FUNCTION_BLOCK basicInfluentFeedLogic (* Basic Function Block Type *)
  (* Standard: 61499-2 *)
  (* Version 0.0, 13/09/2026, Template *)
  PACKAGE Hidryco.HidrycoLib;
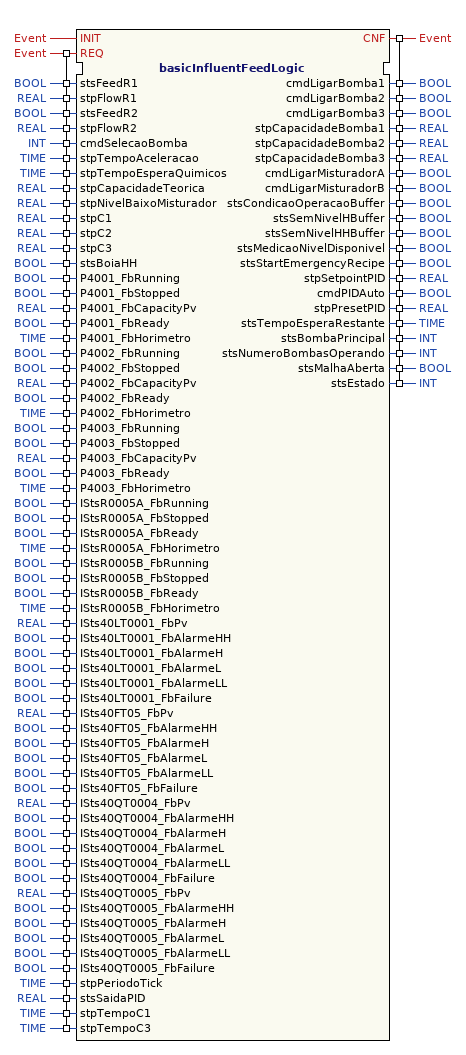
  EVENT_INPUT
    INIT;
    REQ WITH stsFeedR1, stpFlowR1, stsFeedR2, stpFlowR2, cmdSelecaoBomba, stpTempoAceleracao, stpTempoEsperaQuimicos, stpCapacidadeTeorica, stpNivelBaixoMisturador, stpC1, stpC2, stpC3, stsBoiaHH, P4001_FbRunning, P4001_FbStopped, P4001_FbCapacityPv, P4001_FbReady, P4001_FbHorimetro, P4002_FbRunning, P4002_FbStopped, P4002_FbCapacityPv, P4002_FbReady, P4002_FbHorimetro, P4003_FbRunning, P4003_FbStopped, P4003_FbCapacityPv, P4003_FbReady, P4003_FbHorimetro, IStsR0005A_FbRunning, IStsR0005A_FbStopped, IStsR0005A_FbReady, IStsR0005A_FbHorimetro, IStsR0005B_FbRunning, IStsR0005B_FbStopped, IStsR0005B_FbReady, IStsR0005B_FbHorimetro, ISts40LT0001_FbPv, ISts40LT0001_FbAlarmeHH, ISts40LT0001_FbAlarmeH, ISts40LT0001_FbAlarmeL, ISts40LT0001_FbAlarmeLL, ISts40LT0001_FbFailure, ISts40FT05_FbPv, ISts40FT05_FbAlarmeHH, ISts40FT05_FbAlarmeH, ISts40FT05_FbAlarmeL, ISts40FT05_FbAlarmeLL, ISts40FT05_FbFailure, ISts40QT0004_FbPv, ISts40QT0004_FbAlarmeHH, ISts40QT0004_FbAlarmeH, ISts40QT0004_FbAlarmeL, ISts40QT0004_FbAlarmeLL, ISts40QT0004_FbFailure, ISts40QT0005_FbPv, ISts40QT0005_FbAlarmeHH, ISts40QT0005_FbAlarmeH, ISts40QT0005_FbAlarmeL, ISts40QT0005_FbAlarmeLL, ISts40QT0005_FbFailure, stpPeriodoTick, stsSaidaPID, stpTempoC1, stpTempoC3; (* Normal Execution Request *)
  END_EVENT
  EVENT_OUTPUT
    CNF WITH cmdLigarBomba1, cmdLigarBomba2, cmdLigarBomba3, stpCapacidadeBomba1, stpCapacidadeBomba2, stpCapacidadeBomba3, cmdLigarMisturadorA, cmdLigarMisturadorB, stsCondicaoOperacaoBuffer, stsSemNivelHBuffer, stsSemNivelHHBuffer, stsMedicaoNivelDisponivel, stsStartEmergencyRecipe, stpSetpointPID, cmdPIDAuto, stpPresetPID, stsTempoEsperaRestante, stsBombaPrincipal, stsNumeroBombasOperando, stsMalhaAberta, stsEstado; (* Execution Confirmation *)
  END_EVENT
  VAR_INPUT
    stsFeedR1 : BOOL;
    stpFlowR1 : REAL;
    stsFeedR2 : BOOL;
    stpFlowR2 : REAL;
    cmdSelecaoBomba : INT;
    stpTempoAceleracao : TIME; (* Espera antes de controlar as duas bombas juntas *)
    stpTempoEsperaQuimicos : TIME; (* Espera para reiniciar após pH e condutividade normalizarem *)
    stpCapacidadeTeorica : REAL; (* Vazão nominal, para a malha aberta *)
    stpNivelBaixoMisturador : REAL; (* Bloqueio para misturadores *)
    stpC1 : REAL;
    stpC2 : REAL;
    stpC3 : REAL;
    stsBoiaHH : BOOL;
    P4001_FbRunning : BOOL;
    P4001_FbStopped : BOOL;
    P4001_FbCapacityPv : REAL;
    P4001_FbReady : BOOL;
    P4001_FbHorimetro : TIME;
    P4002_FbRunning : BOOL;
    P4002_FbStopped : BOOL;
    P4002_FbCapacityPv : REAL;
    P4002_FbReady : BOOL;
    P4002_FbHorimetro : TIME;
    P4003_FbRunning : BOOL;
    P4003_FbStopped : BOOL;
    P4003_FbCapacityPv : REAL;
    P4003_FbReady : BOOL;
    P4003_FbHorimetro : TIME;
    IStsR0005A_FbRunning : BOOL;
    IStsR0005A_FbStopped : BOOL;
    IStsR0005A_FbReady : BOOL;
    IStsR0005A_FbHorimetro : TIME;
    IStsR0005B_FbRunning : BOOL;
    IStsR0005B_FbStopped : BOOL;
    IStsR0005B_FbReady : BOOL;
    IStsR0005B_FbHorimetro : TIME;
    ISts40LT0001_FbPv : REAL;
    ISts40LT0001_FbAlarmeHH : BOOL;
    ISts40LT0001_FbAlarmeH : BOOL;
    ISts40LT0001_FbAlarmeL : BOOL;
    ISts40LT0001_FbAlarmeLL : BOOL;
    ISts40LT0001_FbFailure : BOOL;
    ISts40FT05_FbPv : REAL;
    ISts40FT05_FbAlarmeHH : BOOL;
    ISts40FT05_FbAlarmeH : BOOL;
    ISts40FT05_FbAlarmeL : BOOL;
    ISts40FT05_FbAlarmeLL : BOOL;
    ISts40FT05_FbFailure : BOOL;
    ISts40QT0004_FbPv : REAL;
    ISts40QT0004_FbAlarmeHH : BOOL;
    ISts40QT0004_FbAlarmeH : BOOL;
    ISts40QT0004_FbAlarmeL : BOOL;
    ISts40QT0004_FbAlarmeLL : BOOL;
    ISts40QT0004_FbFailure : BOOL;
    ISts40QT0005_FbPv : REAL;
    ISts40QT0005_FbAlarmeHH : BOOL;
    ISts40QT0005_FbAlarmeH : BOOL;
    ISts40QT0005_FbAlarmeL : BOOL;
    ISts40QT0005_FbAlarmeLL : BOOL;
    ISts40QT0005_FbFailure : BOOL;
    stpPeriodoTick : TIME;
    stsSaidaPID : REAL;
    stpTempoC1 : TIME;
    stpTempoC3 : TIME;
  END_VAR
  VAR_OUTPUT
    cmdLigarBomba1 : BOOL;
    cmdLigarBomba2 : BOOL;
    cmdLigarBomba3 : BOOL;
    stpCapacidadeBomba1 : REAL;
    stpCapacidadeBomba2 : REAL;
    stpCapacidadeBomba3 : REAL;
    cmdLigarMisturadorA : BOOL;
    cmdLigarMisturadorB : BOOL;
    stsCondicaoOperacaoBuffer : BOOL; (* Operating condition da fase Feed, nos dois reatores. FALSE quando o buffer não pode alimentar *)
    stsSemNivelHBuffer : BOOL;
    stsSemNivelHHBuffer : BOOL;
    stsMedicaoNivelDisponivel : BOOL;
    stsStartEmergencyRecipe : BOOL;
    stpSetpointPID : REAL;
    cmdPIDAuto : BOOL;
    stpPresetPID : REAL;
    stsTempoEsperaRestante : TIME;
    stsBombaPrincipal : INT;
    stsNumeroBombasOperando : INT;
    stsMalhaAberta : BOOL;
    stsEstado : INT;
  END_VAR
  VAR
    iEstado : INT;
    idxDuty1 : INT;
    idxDuty2 : INT;
    tEsperaQuim : TIME;
    tAcel : TIME;
    tC1 : TIME;
    tC3 : TIME;
    bQuimOkAnt : BOOL;
    rSaida : REAL;
  END_VAR
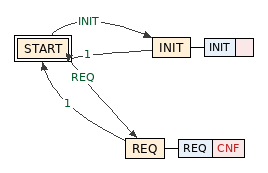
  EC_STATES
    START; (* Initial State *)
    INIT : INIT;
    REQ : REQ -> CNF;
  END_STATES
  EC_TRANSITIONS
    START TO INIT := INIT;
    INIT TO START := 1;
    START TO REQ := REQ;
    REQ TO START := 1;
  END_TRANSITIONS
  ALGORITHM INIT IN ST: (* Initialization algorithm *)
iEstado := 0;
idxDuty1 := 0;
idxDuty2 := 0;
tEsperaQuim := stpTempoEsperaQuimicos;
tAcel := stpTempoAceleracao;
tC1 := stpTempoC1;
tC3 := stpTempoC3;
bQuimOkAnt := FALSE;
rSaida := 0.0;
cmdLigarBomba1 := FALSE; cmdLigarBomba2 := FALSE; cmdLigarBomba3 := FALSE;
stpCapacidadeBomba1 := 0.0; stpCapacidadeBomba2 := 0.0; stpCapacidadeBomba3 := 0.0;
cmdLigarMisturadorA := FALSE; cmdLigarMisturadorB := FALSE;
stsCondicaoOperacaoBuffer := FALSE;
stsSemNivelHBuffer := TRUE;
stsSemNivelHHBuffer := TRUE;
stsMedicaoNivelDisponivel := FALSE;
stsStartEmergencyRecipe := FALSE;
stpSetpointPID := 0.0;
cmdPIDAuto := FALSE;
stpPresetPID := 0.0;
stsTempoEsperaRestante := T#0s;
stsBombaPrincipal := 0;
stsNumeroBombasOperando := 0;
stsMalhaAberta := FALSE;
stsEstado := 0;

;
  END_ALGORITHM
  ALGORITHM REQ IN ST: (* Normally executed algorithm *)
  VAR_TEMP
    bFeedAtivo : BOOL;
    bQuimOk : BOOL;
    bBombaDisp : BOOL;
    bVazaoLL : BOOL;
    bReadyD1 : BOOL;
    bReadyD2 : BOOL;
    rSpBruto : REAL;
    nLigadas : INT;
    idxCand : INT;
    tMenor : TIME;
  END_VAR
stsSemNivelHBuffer := NOT ISts40LT0001_FbAlarmeH;
stsSemNivelHHBuffer := NOT stsBoiaHH;
stsMedicaoNivelDisponivel := NOT ISts40LT0001_FbFailure;
stsStartEmergencyRecipe := ISts40LT0001_FbAlarmeHH
AND NOT ISts40LT0001_FbFailure;
(*------------------------------------------------------------------
2. QUÍMICOS — narrativa 2.2, 2.3.6 e 2.3.7
pH ou condutividade fora de faixa, ou falha de medição de
qualquer um dos dois, param a alimentação.
Temporizador de retomada: conta apenas com AMBOS dentro da
faixa. Qualquer saída de faixa rearma do zero.
------------------------------------------------------------------*)
bQuimOk := NOT ISts40QT0005_FbAlarmeL AND NOT ISts40QT0005_FbAlarmeH
AND NOT ISts40QT0004_FbAlarmeL AND NOT ISts40QT0004_FbAlarmeH
AND NOT ISts40QT0005_FbFailure AND NOT ISts40QT0004_FbFailure;
IF bQuimOk THEN
	IF NOT bQuimOkAnt THEN
		tEsperaQuim := stpTempoEsperaQuimicos; (* borda: arma *)
	ELSIF tEsperaQuim > stpPeriodoTick THEN
		tEsperaQuim := tEsperaQuim - stpPeriodoTick;
	ELSE
		tEsperaQuim := T#0s; (* expirou *)
	END_IF;
ELSE
	tEsperaQuim := stpTempoEsperaQuimicos; (* rearma *)
END_IF;
bQuimOkAnt := bQuimOk;
stsTempoEsperaRestante := tEsperaQuim;
(*------------------------------------------------------------------
3. BOMBAS RODANDO E LL DE VAZÃO
O atraso do alarme é feito pelo bloco de sensor. Aqui só a
supressão: com bomba parada a vazão é zero por definição, e o
alarme não pode bloquear a alimentação.
------------------------------------------------------------------*)
nLigadas := 0;
IF P4001_FbRunning THEN nLigadas := nLigadas + 1; END_IF;
IF P4002_FbRunning THEN nLigadas := nLigadas + 1; END_IF;
IF P4003_FbRunning THEN nLigadas := nLigadas + 1; END_IF;
stsNumeroBombasOperando := nLigadas;
bVazaoLL := (nLigadas > 0)
AND ISts40FT05_FbAlarmeLL
AND NOT ISts40FT05_FbFailure;
(*------------------------------------------------------------------
4. DISPONIBILIDADE — narrativa 1.4.2
------------------------------------------------------------------*)
bBombaDisp := P4001_FbReady OR P4002_FbReady OR P4003_FbReady;
(*------------------------------------------------------------------
5. CONDIÇÃO DE OPERAÇÃO DO BUFFER
Vai para a operating condition da fase Feed dos dois reatores.
Narrativa 2.2: a alimentação para em LL de nível, pH fora de
faixa e condutividade fora de faixa.
------------------------------------------------------------------*)
stsCondicaoOperacaoBuffer := bBombaDisp
AND bQuimOk
AND (tEsperaQuim = T#0s)
AND NOT ISts40LT0001_FbAlarmeLL
AND NOT ISts40LT0001_FbFailure
AND NOT bVazaoLL;
(*------------------------------------------------------------------
6. SETPOINT DE VAZÃO — narrativa 2.2 e 3.2.1
O Nereda envia m³/h; o PI converte em capacidade.
Apenas uma fase Feed pode estar em RUN por vez.
------------------------------------------------------------------*)
bFeedAtivo := stsFeedR1 OR stsFeedR2;
IF stsFeedR1 THEN rSpBruto := stpFlowR1;
ELSIF stsFeedR2 THEN rSpBruto := stpFlowR2;
ELSE rSpBruto := 0.0;
END_IF;
IF rSpBruto < 0.0 THEN rSpBruto := 0.0; END_IF;
stpSetpointPID := rSpBruto;
(*------------------------------------------------------------------
7. ESCOLHA DAS BOMBAS — narrativa 1.4.9
idxCand = próxima candidata: disponível, ainda não comandada,
de MENOR horímetro (FbHorimetro = tempo de operação).
Em modo fixo, a candidata é a bomba escolhida pelo operador.
------------------------------------------------------------------*)
idxCand := 0;
tMenor := T#999999s;
IF cmdSelecaoBomba = 1 THEN
IF P4001_FbReady AND (idxDuty1 <> 1) AND (idxDuty2 <> 1) THEN idxCand := 1; END_IF;
ELSIF cmdSelecaoBomba = 2 THEN
IF P4002_FbReady AND (idxDuty1 <> 2) AND (idxDuty2 <> 2) THEN idxCand := 2; END_IF;
ELSIF cmdSelecaoBomba = 3 THEN
IF P4003_FbReady AND (idxDuty1 <> 3) AND (idxDuty2 <> 3) THEN idxCand := 3; END_IF;
ELSE
IF P4001_FbReady AND (idxDuty1 <> 1) AND (idxDuty2 <> 1)
AND (P4001_FbHorimetro <= tMenor) THEN
idxCand := 1; tMenor := P4001_FbHorimetro;
END_IF;
IF P4002_FbReady AND (idxDuty1 <> 2) AND (idxDuty2 <> 2)
AND (P4002_FbHorimetro < tMenor) THEN
idxCand := 2; tMenor := P4002_FbHorimetro;
END_IF;
IF P4003_FbReady AND (idxDuty1 <> 3) AND (idxDuty2 <> 3)
AND (P4003_FbHorimetro < tMenor) THEN
idxCand := 3; tMenor := P4003_FbHorimetro;
END_IF;
END_IF;
(* Disponibilidade das bombas atualmente comandadas *)
bReadyD1 := FALSE;
CASE idxDuty1 OF
1: bReadyD1 := P4001_FbReady;
2: bReadyD1 := P4002_FbReady;
3: bReadyD1 := P4003_FbReady;
END_CASE;
bReadyD2 := FALSE;
CASE idxDuty2 OF
1: bReadyD2 := P4001_FbReady;
2: bReadyD2 := P4002_FbReady;
3: bReadyD2 := P4003_FbReady;
END_CASE;
stsBombaPrincipal := idxDuty1;
(*------------------------------------------------------------------
8. MÁQUINA DE ESTADOS — narrativa 2.2
0 Parado · 1 Partindo · 2 Uma bomba · 3 Sobe (C2)
4 Duas bombas · 5 Desce · 6 Parando
Na partida não há capacidade fixa: o PI assume desde o início e
a rampa do inversor cuida do transitório. C2 é usado apenas na
transição de uma para duas bombas.
------------------------------------------------------------------*)
CASE iEstado OF
0: (*--- PARADO ---*)
idxDuty1 := 0; idxDuty2 := 0;
cmdPIDAuto := FALSE; stpPresetPID := 0.0; rSaida := 0.0;
tC1 := stpTempoC1; tC3 := stpTempoC3; tAcel := stpTempoAceleracao;
IF bFeedAtivo AND stsCondicaoOperacaoBuffer AND (idxCand <> 0) THEN
idxDuty1 := idxCand;
iEstado := 1;
END_IF;
1: (*--- PARTINDO: comanda a duty, PI já em automático ---*)
cmdPIDAuto := NOT ISts40FT05_FbFailure;
IF NOT bFeedAtivo OR NOT stsCondicaoOperacaoBuffer THEN
iEstado := 6;
ELSIF NOT bReadyD1 THEN
(* Perdeu antes de confirmar: troca direta pela candidata *)
IF idxCand <> 0 THEN idxDuty1 := idxCand;
ELSE idxDuty1 := 0; iEstado := 6;
END_IF;
ELSIF ((idxDuty1 = 1) AND P4001_FbRunning)
OR ((idxDuty1 = 2) AND P4002_FbRunning)
OR ((idxDuty1 = 3) AND P4003_FbRunning) THEN
iEstado := 2;
END_IF;
2: (*--- UMA BOMBA EM CONTROLE ---*)
cmdPIDAuto := NOT ISts40FT05_FbFailure;
idxDuty2 := 0;
IF rSaida >= stpC1 THEN
IF tC1 > stpPeriodoTick THEN tC1 := tC1 - stpPeriodoTick;
ELSE tC1 := T#0s; END_IF;
ELSE
tC1 := stpTempoC1;
END_IF;
IF NOT bFeedAtivo OR NOT stsCondicaoOperacaoBuffer THEN
iEstado := 6;
ELSIF NOT bReadyD1 THEN
(* Troca direta, sem passar pelo Parado *)
IF idxCand <> 0 THEN
idxDuty1 := idxCand;
iEstado := 1; (* aguarda o FbRunning da nova *)
ELSE
idxDuty1 := 0;
iEstado := 6;
END_IF;
ELSIF (tC1 = T#0s) AND (idxCand <> 0) THEN
idxDuty2 := idxCand;
tAcel := stpTempoAceleracao;
iEstado := 3;
END_IF;
3: (*--- SOBE: transição de uma para duas bombas — narrativa 2.2 ---
Única etapa em que C2 é usado. A primeira cai para C2, a
segunda parte em C2, e o PI fica em manual travado nesse
valor durante a aceleração. *)
cmdPIDAuto := FALSE;
stpPresetPID := stpC2;
rSaida := stpC2;
IF tAcel > stpPeriodoTick THEN tAcel := tAcel - stpPeriodoTick;
ELSE tAcel := T#0s; END_IF;
IF NOT bFeedAtivo OR NOT stsCondicaoOperacaoBuffer THEN
iEstado := 6;
ELSIF NOT bReadyD1 THEN
(* A principal caiu durante a transição: a segunda assume *)
idxDuty1 := idxDuty2; idxDuty2 := 0;
tC1 := stpTempoC1;
iEstado := 2;
ELSIF NOT bReadyD2 THEN
idxDuty2 := 0;
tC1 := stpTempoC1;
iEstado := 2;
ELSIF tAcel = T#0s THEN
tC3 := stpTempoC3;
iEstado := 4;
END_IF;
4: (*--- DUAS BOMBAS EM CONTROLE CONJUNTO ---*)
cmdPIDAuto := NOT ISts40FT05_FbFailure;
IF rSaida <= stpC3 THEN
IF tC3 > stpPeriodoTick THEN tC3 := tC3 - stpPeriodoTick;
ELSE tC3 := T#0s; END_IF;
ELSE
tC3 := stpTempoC3;
END_IF;
IF NOT bFeedAtivo OR NOT stsCondicaoOperacaoBuffer THEN
iEstado := 6;
ELSIF NOT bReadyD1 THEN
(* Perdeu a principal: a segunda passa a ser a principal *)
idxDuty1 := idxDuty2;
IF idxCand <> 0 THEN
idxDuty2 := idxCand;
tAcel := stpTempoAceleracao; (* recontado do início *)
iEstado := 3;
ELSE
idxDuty2 := 0;
tC1 := stpTempoC1;
iEstado := 2;
END_IF;
ELSIF NOT bReadyD2 THEN
IF idxCand <> 0 THEN
idxDuty2 := idxCand;
tAcel := stpTempoAceleracao; (* recontado do início *)
iEstado := 3;
ELSE
idxDuty2 := 0;
tC1 := stpTempoC1;
iEstado := 2;
END_IF;
ELSIF tC3 = T#0s THEN
iEstado := 5;
END_IF;
5: (*--- DESCE: volta para uma bomba ---
Sai a que está em operação há mais tempo, ou seja, a
primeira que entrou — narrativa 1.4.9. *)
idxDuty1 := idxDuty2;
idxDuty2 := 0;
tC1 := stpTempoC1;
iEstado := 2;
6: (*--- PARANDO ---*)
idxDuty1 := 0; idxDuty2 := 0;
cmdPIDAuto := FALSE; stpPresetPID := 0.0; rSaida := 0.0;
IF nLigadas = 0 THEN
iEstado := 0;
END_IF;
END_CASE;
stsEstado := iEstado;
(*------------------------------------------------------------------
9. CAPACIDADE — narrativa 2.2
Falha do medidor: converte o setpoint em capacidade pela
capacidade teórica (malha aberta).
Nos estados 3, 5 e 6 a capacidade já foi definida pelo estado.
------------------------------------------------------------------*)
IF ISts40FT05_FbFailure AND (iEstado >= 1) AND (iEstado <= 4) THEN
stsMalhaAberta := TRUE;
IF stpCapacidadeTeorica > 0.0 THEN
IF idxDuty2 <> 0 THEN
rSaida := 100.0 * stpSetpointPID / (2.0 * stpCapacidadeTeorica);
ELSE
rSaida := 100.0 * stpSetpointPID / stpCapacidadeTeorica;
END_IF;
ELSE
rSaida := 0.0;
END_IF;
IF rSaida > 100.0 THEN rSaida := 100.0; END_IF;
stpPresetPID := rSaida; (* mantém o PI acompanhando *)
ELSE
stsMalhaAberta := FALSE;
IF (iEstado = 1) OR (iEstado = 2) OR (iEstado = 4) THEN
rSaida := stsSaidaPID;
END_IF;
END_IF;
(*------------------------------------------------------------------
10. COMANDOS DAS BOMBAS
Derivados de idxDuty1 e idxDuty2 — fonte única, sem comando
espalhado pelos estados. A capacidade é a MESMA para todas as
bombas em operação (narrativa 2.2).
------------------------------------------------------------------*)
cmdLigarBomba1 := (idxDuty1 = 1) OR (idxDuty2 = 1);
cmdLigarBomba2 := (idxDuty1 = 2) OR (idxDuty2 = 2);
cmdLigarBomba3 := (idxDuty1 = 3) OR (idxDuty2 = 3);
stpCapacidadeBomba1 := 0.0;
stpCapacidadeBomba2 := 0.0;
stpCapacidadeBomba3 := 0.0;
IF cmdLigarBomba1 THEN stpCapacidadeBomba1 := rSaida; END_IF;
IF cmdLigarBomba2 THEN stpCapacidadeBomba2 := rSaida; END_IF;
IF cmdLigarBomba3 THEN stpCapacidadeBomba3 := rSaida; END_IF;
(*------------------------------------------------------------------
11. MISTURADORES — narrativa 2.3.2
Em automático operam continuamente. Nível baixo e LL são
condição de Ready do próprio misturador — não duplicar
intertravamento aqui.
------------------------------------------------------------------*)
cmdLigarMisturadorA := TRUE;
cmdLigarMisturadorB := TRUE;
;
  END_ALGORITHM
END_FUNCTION_BLOCK
